(* CoDeSys 2.3 library: ClientStrSock.lib *)
(* Libraries: TcBase.lib 14.5.09 12:14:08, TcSystem.lib 10.9.09 12:54:20, STANDARD.LIB 5.6.98 12:03:02, TcpIp.lib 13.10.11 10:31:34, TcUtilities.lib 17.9.09 15:40:48, TcSocketHelper.lib 20.8.09 10:46:08 *)

(* Global variable list: Global_Variables *)
VAR_GLOBAL CONSTANT
	PLCPRJ_MAX_CONNECTIONS					: UDINT := 5;(* Max. number of server<->client connections *)
	PLCPRJ_SERVER_RESPONSE_TIMEOUT		: TIME 	:= T#500ms;
	PLCPRJ_CLIENT_SEND_CYCLE_TIME			: TIME 	:= T#500ms;

	PLCPRJ_RECEIVER_POLLING_CYCLE_TIME		: TIME 	:= T#200ms;
	PLCPRJ_BUFFER_SIZE						: UDINT := 1000;(* Max. internal fifo/receiver buffer size *)

	(* Some project specific error codes *)
	PLCPRJ_ERROR_RECEIVE_BUFFER_OVERFLOW	: UDINT := 16#8101; (* receive fifo/buffer overflow*)
	PLCPRJ_ERROR_SEND_BUFFER_OVERFLOW		: UDINT := 16#8102;(* send fifo/buffer overflow *)
	PLCPRJ_ERROR_RESPONSE_TIMEOUT			: UDINT := 16#8103;(* receive timeout error *)

	MSG_HEADER 									: STRING(10) :=	'#STR.HEAD#';
	MSG_DATA 										: STRING(10) :=  	'#STR.DATA#';

	MSG_TYPE_SET									: STRING(10) :=	'SET0000000'		;
	MSG_TYPE_RESET								: STRING(10) :=	'RESET00000'	;
	MSG_TYPE_MONITORING							: STRING(10) := 	'MONITOR000'	;

	MSG_SYSTEM_TYPE_1							: STRING(10) := 	'LIGHT00000'	;
	MSG_SYSTEM_TYPE_2							: STRING(10) := 	'ENERGY0000'	;
	MSG_SYSTEM_TYPE_3							: STRING(10) := 	'LEAKAGE000'	;
	MSG_SYSTEM_TYPE_4							: STRING(10) :=	'CLIMATE000'	;

	MSG_DATA_TYPE_1DIGIT							: STRING(10) := 	'1DIG000000'	;
	MSG_DATA_TYPE_3DIGIT							: STRING(10) := 	'3DIG000000'	; (* данные отмасштабированы в пределах 0-255 по шкале 0-100*)
	MSG_DATA_TYPE_4DIGIT							: STRING(10) := 	'4DIG000000'	;
	MSG_DATA_TYPE_8DIGIT							: STRING(10) := 	'8DIG000000'	;
	MSG_DATA_TYPE_S								: STRING(10) :=	'STRING0000'	;

	ARR_DATA_SIZE_1D								: INT := 128;
	ARR_DATA_SIZE_3D								: INT := 32;
	ARR_DATA_SIZE_4D								: INT := 32;
	ARR_DATA_SIZE_8D								: INT := 16;
	ARR_DATA_SIZE_S								: INT := 128;

	TO_SEND										:BYTE:=4;
	TO_RECEIVE									:BYTE :=128;

(*
header
msgMsgType  		= get_buffer_string(strData, 10);
    msgSystemType 		= get_buffer_string(strData, 10);
    msgDeviceType		= get_buffer_string(strData, 10);
    msgDevNum 			= get_buffer_string(strData, 10);
    msgDataType 		= get_buffer_string(strData, 10);
    msgDevision 		= get_buffer_string(strData, 10);
    msgSubDev	 		= get_buffer_string(strData, 10);
    msgReserved_1 		= get_buffer_string(strData, 10);
    msgReserved_2 		= get_buffer_string(strData, 10);
dataheader
*)
(*

MSG_HEADER 				= '#STR.HEAD#'	;
MSG_DATA 				= '#STR.DATA#'	;

MSG_TYPE_SET				= 'SET'		;
MSG_TYPE_RESET				= 'RESET'	;
MSG_TYPE_MONITORING			= 'MONITOR'	;

MSG_SYSTEM_TYPE_1			= 'LIGHT'	;
MSG_SYSTEM_TYPE_2			= 'ENERGY'	;
MSG_SYSTEM_TYPE_3			= 'LEAKAGE'	;
MSG_SYSTEM_TYPE_4			= 'CLIMATE'	;

MSG_DATA_TYPE_1DIGIT			= '1DIG'	;
MSG_DATA_TYPE_3DIGIT			= '3DIG'	;
MSG_DATA_TYPE_4DIGIT			= '4DIG'	;
MSG_DATA_TYPE_150DIGIT			= 'STRING'	;

*)
END_VAR
VAR_GLOBAL
	random		: DRAND := (seed := 10);(* random number generator *)
END_VAR

(* POU F_ADSLOGERROR, ST *)
FUNCTION F_ADSLOGERROR : DINT
(* This function logs communication error messages to the TwinCAT System Log View *)
VAR_INPUT
	sPrefix		: STRING(20);(* Debug message prefix string (allows the identification of log message source) *)
	nErrID		: DWORD; (* Error code *)
END_VAR
IF nErrId = 0 THEN
	F_ADSLOGERROR := ADSLOGSTR( ADSLOG_MSGTYPE_HINT OR ADSLOG_MSGTYPE_LOG, CONCAT( sPrefix, ' No error!   %s'),'' );
ELSIF (  nErrId AND DWORD#16#80000000 ) = 16#80000000 THEN
	F_ADSLOGERROR := ADSLOGDINT( ADSLOG_MSGTYPE_ERROR OR ADSLOG_MSGTYPE_LOG, CONCAT( sPrefix, ' Win32 error: %d' ), SCODE_CODE( nErrId ) );
ELSIF (nErrId AND 16#00008100) =16#00008100 THEN
	F_ADSLOGERROR := ADSLOGDINT( ADSLOG_MSGTYPE_ERROR OR ADSLOG_MSGTYPE_LOG, CONCAT( sPrefix, ' Internal PLC sample project (user) error: %d' ), nErrId );
ELSIF (nErrId AND 16#00008000) =16#00008000 THEN
	F_ADSLOGERROR := ADSLOGDINT( ADSLOG_MSGTYPE_ERROR OR ADSLOG_MSGTYPE_LOG, CONCAT( sPrefix, ' Internal TCP/IP Connection Server error: %d' ), nErrId );
ELSE
	F_ADSLOGERROR := ADSLOGDINT( ADSLOG_MSGTYPE_ERROR OR ADSLOG_MSGTYPE_LOG, CONCAT( sPrefix, ' TwinCAT System error: %d' ), nErrId );
END_IF
END_FUNCTION

(* POU SCODE_CODE, ST *)
FUNCTION SCODE_CODE : DWORD
(* Helper function: returns the lower word of error code *)
VAR_INPUT
	sc		: UDINT;
END_VAR
SCODE_CODE := 16#FFFF AND UDINT_TO_DWORD( sc );
END_FUNCTION

(* POU F_ADSLOGSTRING, ST *)
FUNCTION F_ADSLOGSTRING : DINT
(* This function logs message string to the TwinCAT System Log View *)
VAR_INPUT
	sPrefix	: STRING(20);(* Debug message prefix string (allows the identification of log message source) *)
	sMsg	: T_MaxString;(* Message string *)
END_VAR
VAR
END_VAR
F_ADSLOGSTRING := ADSLOGSTR( ADSLOG_MSGTYPE_HINT OR ADSLOG_MSGTYPE_LOG, CONCAT( sPrefix, '%s' ), sMsg );
END_FUNCTION

(* POU F_DataPrep, ST *)
FUNCTION F_DataPrep : T_MaxString
VAR_INPUT
	msgheader			:STRING(10);
	msgMsgType  		:STRING(10);
	msgSystemType 		:STRING(10);
	msgDeviceType		:STRING(10);
    	msgDevNum 			:STRING(10);
    	msgDataType 		:STRING(10);
    	msgDevision 			:STRING(10);
    	msgSubDev	 		:STRING(10);
    	msgReserved_1 		:STRING(10);
    	msgReserved_2 		:STRING(10);
	dataheader			:STRING(10);
	data1dig				: ARRAY[0..ARR_DATA_SIZE_1D] OF INT;
	data3dig				: ARRAY[0..ARR_DATA_SIZE_3D] OF INT;
	data3dig_Htr			: INT:=255;
	data3dig_Ltr			: INT:=0;
	data4dig				: ARRAY[0..ARR_DATA_SIZE_4D] OF INT;
	data8dig				: ARRAY[0..ARR_DATA_SIZE_8D] OF DINT;
	dataS				: STRING(128);


END_VAR
VAR
	i,j : INT;
	str: T_MaxString	:= '';
	str2: STRING(128) := '';
	str3: STRING(3)	:= '10';
	value:  DINT;
END_VAR
str:= CONCAT(str, msgheader);
str:= CONCAT(str, msgMsgType);
str:= CONCAT(str, msgSystemType);
str:= CONCAT(str, msgDeviceType);
str:= CONCAT(str, msgDevNum);
str:= CONCAT(str, msgDataType);

str:= CONCAT(str, msgDevision);
str:= CONCAT(str, msgSubDev);
str:= CONCAT(str, msgReserved_1);
str:= CONCAT(str, msgReserved_2);
str:= CONCAT(str, dataheader);

IF msgDataType = MSG_DATA_TYPE_1DIGIT THEN

		FOR i:=0 TO ARR_DATA_SIZE_1D-1 DO
			IF data1dig[i] = 1 THEN
				MEMCPY(ADR(str)+110+i, ADR(str3),1);
			ELSE
				MEMCPY(ADR(str)+110+i, ADR(str3)+1,1);
			END_IF
		END_FOR
		MEMSET(ADR(str)+110+ ARR_DATA_SIZE_1D, 33, 255 - (110+ ARR_DATA_SIZE_1D) ); 	(* заполняем восклицательными знаками остаток сообщения*)
END_IF




IF msgDataType = MSG_DATA_TYPE_3DIGIT THEN
		FOR i:=0 TO ARR_DATA_SIZE_3D-1 DO
			value:= F_ValScale( data3dig[i], data3dig_Htr, data3dig_Ltr);
			str2:= F_ValToStr(value, 3);
			MEMCPY(ADR(str)+110+i*3, ADR(str2), 3);
		END_FOR
		MEMSET(ADR(str)+110+ ARR_DATA_SIZE_3D*3, 33, 255 - (110+ ARR_DATA_SIZE_3D*3) ); 	(* заполняем восклицательными знаками остаток сообщения*)
END_IF




IF msgDataType = MSG_DATA_TYPE_4DIGIT THEN

		FOR i:=0 TO ARR_DATA_SIZE_4D-1 DO
			str2:= F_ValToStr(data4dig[i], 4);
			MEMCPY(ADR(str)+110+i*4, ADR(str2), 4);
		END_FOR
		MEMSET(ADR(str)+110+ ARR_DATA_SIZE_4D*4, 33, 255 - (110+ ARR_DATA_SIZE_4D*4) ); 	(* заполняем восклицательными знаками остаток сообщения*)
END_IF

IF msgDataType = MSG_DATA_TYPE_8DIGIT THEN
		FOR i:=0 TO ARR_DATA_SIZE_8D-1 DO
			str2:= F_ValToStr(data8dig[i], 8);
			MEMCPY(ADR(str)+110+i*8, ADR(str2), 8);
		END_FOR
		MEMSET(ADR(str)+110+ ARR_DATA_SIZE_8D*8, 33, 255 - (110+ ARR_DATA_SIZE_8D*8) ); 	(* заполняем восклицательными знаками остаток сообщения*)
END_IF

IF msgDataType = MSG_DATA_TYPE_S  THEN
		MEMCPY(ADR(str)+110, ADR(dataS), 128); 	(* заполняем восклицательными знаками остаток сообщения*)
		MEMSET(ADR(str)+110+128, 33, 255 - (110+ 128) ); 	(* заполняем восклицательными знаками остаток сообщения*)
END_IF

MEMSET(ADR(str)+255, 0, 1); 	(* ставим 0 в самом конце*)
F_DataPrep:=str;
END_FUNCTION

(* POU F_ValScale, ST *)
FUNCTION F_ValScale : DINT
VAR_INPUT
	value : DINT;
	trs_H: INT;
	trs_L: INT;
END_VAR
VAR
	v: INT;
END_VAR

(*
Функция выдает на выходе значение 0 - 100
Аргументами являются входная переменная и верхнее и нижнее значения диапазона
Если входная переменная больше верхнего предела, на выходе 100
Если меньше нижнего предела 0
*)
IF value>trs_H THEN value:= trs_H; END_IF
IF value<trs_L THEN value:= trs_L; END_IF
F_ValScale:= 67;
F_ValScale:= (value - trs_L)*100 / (trs_H - trs_L);
END_FUNCTION

(* POU F_ValToStr, ST *)
FUNCTION F_ValToStr : STRING
VAR_INPUT
	value: DINT; (* значение, которое необходимо перевести в строку*)
	digit: INT; (* количество разрядов, которое должно быть в строчном представлении. Все "пустые" разряды заполняются 0 *)
END_VAR
VAR
	i		: INT := 0;
	val 		: DINT := 0;
	dig		: INT := 0;
	str1		: STRING;
	str2		: STRING;
	str3		: STRING(3):= '000';
END_VAR
IF value <> 0 THEN
val:= value;
	REPEAT
		val := val / 10;
		dig:= dig+1;
	UNTIL
		val = 0
	END_REPEAT
END_IF

str2:= DINT_TO_STRING(value);

FOR i:=0 TO (digit-dig-1) DO
	MEMCPY(ADR(str1)+i, ADR(str3), 1);
END_FOR

MEMCPY(ADR(str1)+digit-dig, ADR(str2), dig);

F_ValToStr:= str1;
END_FUNCTION

(* POU FB_ClientApplication, ST *)
FUNCTION_BLOCK FB_ClientApplication
(* Sample client application. Adapt this code to match your needs. *)

(*
Этот модуль получился аттавизмом. В исходном варианте (который предоставил Бэкхофф) предполагалось, что пользовательская
обработка сообщений будет располагаться прямо здесь. У меня она находится выше - в основной программе. Оттуда вызыва-
ется функция компановки сообщения F_DataPrep и там же определяется когда вызывать отправку. Бэкхофф расчитывал что
я буду писать это здесь... но не сложилось... Пока разбирался, постепенно отключал все лишнее... и в итоге переписал его в
таком виде, в каком он сейчас. Исходный вид (ну или очень близкий к нему ;) ) приведен в комментированом виде ниже.
*)
VAR_INPUT
	bDbg		: BOOL 			:= TRUE;(* TRUE => Enable debug output, FALSE => Disable *)
	sRemoteHost	: STRING(15)	 	:= '127.0.0.1';
	nRemotePort	: UDINT 			:= 9999;
	bEnable		: BOOL 			:= FALSE;
	bRequest	: BOOL:=FALSE;
	msgToServer	: T_MaxString		:= '';
	state: BYTE;
	send_status_reset	:BOOL := FALSE;
END_VAR
VAR_OUTPUT
	eState		: E_SocketConnectionState := eSOCKET_DISCONNECTED;(* TCP/IP connection state *)
	answer		: T_MaxString		:= '';
	bDataReady	: BOOL:= FALSE;
	receive_ok 	: BOOL := FALSE;
	send_ok 		: BOOL:= FALSE;
END_VAR
VAR
	lengthS1		: INT;
	lengthS2		: INT;
	sToServer	: T_MaxString	:= '';
	sFromServer	: T_MaxString	:= '';
	fbClient		: FB_LocalClient;(* Client data exchange control function block *)
	tx 			: FB_FrameStringFifo;(* Tx fifo *)
	rx 			: FB_FrameStringFifo;(* Rx fifo *)
	errors		: FB_ProtErrorFifo;(* Error fifo *)
	sndTimer	: TON;
	rcvTimer		: TON;
(*	state		: BYTE;(* application state *)*)
END_VAR
(*-------------------------- trigger data exchange -----------------------------------------------*)
(*запускаем модуль клиент, передавая сверху в него параметры....*)
fbClient(  bDbg := bDbg, rx := rx, tx := tx, errors := errors, bEnable := bEnable, sRemoteHost := sRemoteHost, nRemotePort := nRemotePort, eState=>eState, received_string=>answer );

(*IF send_status_reset = TRUE THEN send_ok := FALSE; END_IF*)

CASE state OF
	TO_SEND:
		IF fbClient.eState = eSOCKET_CONNECTED THEN
			sToServer := msgToServer;
			tx.A_AddTail( putValue := sToServer );		(* put string to the tx fifo *)
				send_ok:=FALSE;
				IF tx.bOk THEN(* success *)
					send_ok:=TRUE;
				ELSE
					send_ok:=FALSE;
				END_IF

		END_IF

	TO_RECEIVE:
			receive_ok:= FALSE;
			rx.A_RemoveHead();(* fetch string from rx fifo *)
			IF rx.bOk THEN(* success *)
				sFromServer := rx.getValue;
				(* TODO: Check if the response string == request string *)
				receive_ok:= TRUE;
			ELSE
				receive_ok:= FALSE;
			END_IF
END_CASE







(*--------------------------Simple TCP/IP application-----------------------------------------------*)
(* Данный модуль в
state == 0 сбрасывает таймер отправки  и таймаут приема
state == 1 если подключены, взводим таймер отправки сообщения. Если соединения нет уходим в 0:
Пока таймер не сработал крутимся в этом case. Как только таймер сработал
Сбрасываем его
обновляем строку для отправки
вкладываем строку в tx fifo и если это происходит удачно, сбрасываем таймаут приема и переходим в 2:
в противном случае пишем ошибку и остаемся.
state == 2 
Цикл
(
	вырезаем со сдвигом из fifo буфера самое старое сообщение. Если удачно, то  вероятно getvalue(?)
	каким-то образом копируем его в sFromServer и возвращаемся в 0: .Если неудачно, взводим таймаут на прием
	И до тех пор, пока он не случился, крутимся в этом цикле. Если он случился, (!) непонятно (!) у нас все равно
	не наступает условий для выхода из цикла. Условием выхода является упешное извлечение из fifo(rx.bOk). Очень странно... 
	и в таком виде может быть черевато уходами в себя.
)


*)

(*
CASE state OF
	0:(* init state *)
		sndTimer( IN := FALSE, PT := PLCPRJ_CLIENT_SEND_CYCLE_TIME );
		rcvTimer( IN := FALSE, PT := PLCPRJ_SERVER_RESPONSE_TIMEOUT );
		state := 1;

	1:

		(* send string to server *)
		IF fbClient.eState = eSOCKET_CONNECTED THEN
			sndTimer( IN := TRUE );
			IF sndTimer.Q THEN
				sndTimer( IN := FALSE );

				random( );(* create new random number *)
				(*sToServer := CONCAT( 'Random message from client: ', LREAL_TO_STRING(random.Num) );(* simulate user data (string message) *)*)
				lengthS1:= SIZEOF(msgToServer);
				sToServer := msgToServer;
				lengthS2:= SIZEOF(sToServer);


		(*		sToServer := '1234567890123456789012345678901234567890123456789012345678901234567890123456789012345678901234567890AAAAAAAAAA1234567890123456789012345678901234567890123456789012345678901234567890123456789012345678901234567890BBBBBBBBBB123456789012345678901234567890CCCC';
*)
				tx.A_AddTail( putValue := sToServer );(* put string to the tx fifo *)
				IF tx.bOk THEN(* success *)
					rcvTimer( IN := FALSE );
					state := 2;(* wait for response (ECHO from server) ) *)
				ELSE(* TX fifo overflow => log error *)
					errors.A_AddTail( putError := PLCPRJ_ERROR_SEND_BUFFER_OVERFLOW );
				END_IF

			END_IF
		ELSE
			state := 0;
		END_IF

	2:(* wait for response from server *)
		REPEAT
			rx.A_RemoveHead();(* fetch string from rx fifo *)
			IF rx.bOk THEN(* success *)
				sFromServer := rx.getValue;
				(* TODO: Check if the response string == request string *)


				state := 0;(* repeat send-receive cycle *)
			ELSE
				rcvTimer( IN := TRUE );
				IF rcvTimer.Q THEN(* receive timeout => log error *)
					rcvTimer( IN := FALSE );
					errors.A_AddTail( putError := PLCPRJ_ERROR_RESPONSE_TIMEOUT );
					state := 0;
				END_IF
			END_IF
		UNTIL NOT rx.bOk
		END_REPEAT


END_CASE


(*------------------------------- get error messages from error fifo ------------------------------------------*)
(*Отдельный цикл извлекания со сдвигом ошибок из  fifo*)
(*вероятно, bOk - это флаг опустошения буфера... тогда сказанное выше по поводу опасности
 отменяется. Его можно убрать нах. это пока не нужно.
*)
REPEAT
	errors.A_RemoveHead( bDbg := bDbg );
	IF errors.bOk THEN
		;(* TODO: Implement error handler *)
	END_IF
UNTIL NOT errors.bOk
END_REPEAT


*)
END_FUNCTION_BLOCK

(* POU FB_LocalClient, ST *)
FUNCTION_BLOCK FB_LocalClient
(*
----------------------------
НАЗНАЧЕНИЕ
	Устанавливает связь и следит за ее наличием. Передает сообщения. Проверяет входящие.
---------------------------

---------------
Особенности:
	Меня настораживает работа fifo буферов (rx и tx)
	Если передача более или менее работает, то прием сообщений то глючит, то вообще не работает. 
	Пришлось дописать MEMCPY( ADR(received_string), ADR(buffer),  SIZEOF(received_string) ); и только 
	тогда стало появляться приходящее сообщение в received string.

	С отправкой тоже чудеса. Если открыть один сокет и слать пакет скажем раз в секунду, он всегда доходит.
	Если (как в нашем случае) открыть 4 сокета и раз в 300мс слать разные пакеты, то одни не доходят, а других
	приходит (почему-то) лишнее количество... Причем связано это не с какими-то конкретными пакетами. Если 
	поменять их местами в очередности, или даже перезагрузить конечный контроллер, то доходить будут другие.
	Мне не удалось понять где баг. В первую очередь грешу на fifo, т.к. очевидно что здесь что-то не работает...
	Возможно где-то еще есть сюрпизы. 

---------------
*)


VAR_IN_OUT
	tx 			: FB_FrameStringFifo;(* TX fifo *)
	rx 			: FB_FrameStringFifo;(* RX fifo *)
	errors		: FB_ProtErrorFifo;(* Error message fifo *)
END_VAR
VAR_INPUT
	bDbg		: BOOL 			:= TRUE;(* TRUE => Enable debug output, FALSE => Disable debug output *)
	sRemoteHost	: STRING(15) 		:= '192.168.3.229';(* IP address of remote server *)
	nRemotePort	: UDINT			:= 8888;(* Remote server port *)
	bEnable		: BOOL			:= FALSE;(* TRUE => Enable/connect, FALSE => Disable/disconnect *)
	tReconnect	: TIME 			:= T#45s;(* Try to reconnect after this time *)
(*	bRequest: BOOL:= FALSE;*)
END_VAR
VAR_OUTPUT
	eState		: E_SocketConnectionState := eSOCKET_DISCONNECTED;(* TCP/IP connection state *)
	received_string: T_MaxString;
(*	bDataReady: BOOL:=FALSE;*)
END_VAR
VAR
	fbConnect 	: FB_ClientServerConnection := ( tReconnect := T#45s );(* create/release TCP/IP connection *)
	fbSend		: FB_SocketSend;(* send TCP/IP data *)
	fbReceive	: FB_SocketReceive;(* receive TCP/IP data *)
	state 		: BYTE;(* global state *)
	tx_state 		: BYTE;(* tx state *)
	rx_state 		: BYTE;(* rx state *)
	bDisconnect	: BOOL;(* disconnect flag, if set the socket will be closed *)
	pollTimer	: TON;
	cbReceived	: UDINT;(* count of received data bytes *)
	cbRx		: UDINT;(* byte length of received string *)
	rxFrame		: T_MaxString;
	txFrame		: T_MaxString;
	buffer		: ARRAY[0..PLCPRJ_BUFFER_SIZE] OF BYTE;(* Temp. RX buffer *)
	i			: UDINT;
	bAbort		: BOOL;
	sID			: STRING(20) := '';

	bWaitForAnswer: BOOL:=FALSE;
END_VAR
(*
----------------------------
ОПИСАНИЕ (подробное)
---------------------------
state == 0
Сбрасываем fifo приема, передачи и ошибок. Сбрасываем состояния приема и передачи в 0. 
Сбрасываем кол-во принятых данных в 0. Сбрасываем poll таймер. Переходим в state == 1

state == 1
запускаем функциональный блок fbConnect (видимо устанавливаем подключение) крутимся здесь
пока оно не установится. Когда устанавливается, переходим в 2:
state == 2 
Если дизактивирован блок или клиент отключен(поднят флаг), при условии отсутствия входящих и исходящих данных, переходим в 3:
В противном случае  заходим по очереди в ветвления tx_state, rx_state
		tx_state == 0
		Если клиент подключен, извлекаем из tx fifo txFrame. Запускаем блок fbSend со строкой txFrame и, если удачно (bOk), 
		переходим в 1:
		tx_state == 1
		выключаем флаг исполнения  fbSend и проверяем, закончил ли этот блок исполняться (на отправку вписано 5 секунд), если закончил, уходим в 0:
		если при этом были ошибки, делаем дисконнект.

		rx_state == 0
		Если нет дисконнекта, взводим pollTimer, а когда он срабатывает
		Проверяем, (вроде бы) есть ли свободное место в fifo. Если есть, то сбрасываем таймер и выполняем
		блок fbReceive, после чего переходим в 1:
		rx_state == 1
		выключаем флаг исполнения fbReceive и если он закончил работу(на прием так же 5 сек), переходим в  0: а так же
		если не было ошибок и размер принятых данных > 0 (если же принято меньше, то устанавливаем длительность polTimer нормальной)(если были ошибки  пишем их в error fifo и  делаем дисконнект)
		увеличиваем частоту обработки ветвления rx_state, уменьшая до нуля pollTimer
		увеличиваем общий счетчик принятых данных

 		здесь моя вставка копирования из буфера строки

		Далее начинаем цикл (вроде бы парсинга приходящей строки)
		(
			включаем флаг bAbort
			если общее кол-во принятых данных > 0 
			пробегаемся по каждому байту буфера, сравнивая его с 0
			Если находим 0
			запоминаем размер строки + 1 байт знака конца строки
			копируем из буфера в rxFrame данную строку (а если она не лезет, то копируем сколько влезет)
			пихаем rxFrame в rx fifo
			Если успешно (rx.bOk) то сдвигаем значения в буфере на размер забраной строки
				Если в rx fifo есть еще место под rxFrame выключаем флаг bAbort
			Если были ошибки пишем их в eror fifo и делаем дисконнект

			Выходим из цикла если флаг bAbort включен
		)

state == 3
 выключаем блок fbConect и переходим в 0:
---------------------
*)


CASE state OF
	0:(* init state *)
		rx.A_Reset( bDbg := bDbg );(* reset RX fifo (optional) *)
		tx.A_Reset( bDbg := bDbg );(* reset TX fifo (optional) *)
		errors.A_Reset( bDbg := bDbg );(* reset error fifo (optional) *)
		tx_state 		:= 0;
		rx_state 		:= 0;
		pollTimer( IN := FALSE, PT := PLCPRJ_RECEIVER_POLLING_CYCLE_TIME );
		bDisconnect 	:= FALSE;
		cbReceived 	:= 0;
		state 		:= 1;

	1:(* connect *)
		fbConnect( 	sSrvNetID 		:= '',
					nMode			:= CONNECT_MODE_ENABLEDBG,(* enable debug output *)
					sRemoteHost 	:= sRemoteHost,
					nRemotePort 		:= nRemotePort,
					bEnable			:= bEnable,
					tReconnect		:= tReconnect,
					eState			=> eState );
		IF NOT fbConnect.bBusy THEN

			sID 			:= CONCAT( CONCAT('[', DWORD_TO_HEXSTR(fbConnect.hSocket.handle, 4, FALSE) ), ']' );
			tx.sDesc		:= CONCAT( 'CLI.Tx', sID );
			rx.sDesc 		:= CONCAT( 'CLI.Rx', sID );
			errors.sDesc	:= CONCAT( 'CLI.Err', sID );

			IF NOT fbConnect.bError THEN
				IF eState = eSOCKET_CONNECTED THEN(* we are conencted *)
					(*IF bRequest = TRUE THEN*)
					state := 2;
					(*END_IF*)
				END_IF
			ELSE(* connect error => log error *)
				errors.A_AddTail( putError := fbConnect.nErrId );
			END_IF
		END_IF


	2:(* data exchange state *)
		(*bRequest:= FALSE;
		bWaitForAnswer:= TRUE;*)
		bDisconnect := NOT bEnable OR bDisconnect;(* user/internal disconnect requested? *)
		IF bDisconnect AND (tx_state = 0) AND (rx_state = 0) THEN
			state := 3;(* disconnect *)
		ELSE

			(* send tx data *)
			CASE tx_state OF
				0:
					IF NOT bDisconnect THEN
						tx.A_RemoveHead( bDbg := bDbg, getValue => txFrame );(* remove oldest string entry s*)
						IF tx.bOk THEN(* success *)
							fbSend( bExecute := FALSE );
							fbSend(	sSrvNetID 	:= '',
									hSocket		:= fbConnect.hSocket,
									cbLen		:= LEN( txFrame ) + 1,(* send string inclusive string (null) delimiter! *)
									pSrc		:= ADR( txFrame ),(* address of the string variable *)
									bExecute	:= TRUE,
									tTimeout 		:= T#5s );
							tx_state := 1;
						END_IF
					END_IF
				1:(* wait until send not busy *)
					fbSend( bExecute := FALSE );
					IF NOT fbSend.bBusy THEN
						tx_state := 0;
						IF fbSend.bError THEN(* send error => log error and disconnect *)
							errors.A_AddTail( putError := fbSend.nErrId );
							bDisconnect := TRUE;(* set flag *)
						END_IF
					END_IF
			END_CASE



			(* get rx data *)
			CASE rx_state OF
				0:
				(*IF bWaitForAnswer = TRUE THEN*)

					IF NOT bDisconnect THEN
						pollTimer( IN := TRUE );
						IF pollTimer.Q THEN
							IF rx.cbFree >= SIZEOF(rxFrame) THEN(* check free rx fifo space *)
								pollTimer( IN := FALSE );

								fbReceive( bExecute := FALSE );
								fbReceive( 	sSrvNetId	:= '',
											hSocket		:= fbConnect.hSocket,
											cbLen		:= SIZEOF(buffer),(* - cbReceived,*)
											pDest		:= ADR(buffer), (*+ cbReceived,*)
											bExecute	:= TRUE,
											tTimeout		:= T#5s );
								rx_state := 1;
							END_IF
						END_IF
					END_IF
			(*	END_IF*)
				1:(* wait until receive not busy *)
					fbReceive( bExecute := FALSE );
					IF NOT fbReceive.bBusy THEN
						rx_state := 0;
						IF NOT fbReceive.bError THEN
							IF fbReceive.nRecBytes > 0 THEN
								pollTimer( PT := T#0s );(* increase polling speed *)
								cbReceived := cbReceived + fbReceive.nRecBytes;


									MEMSET(ADR(received_string), 0,  SIZEOF(received_string));
									MEMCPY( ADR(received_string), ADR(buffer),  SIZEOF(received_string) );
									(*bWaitForAnswer:= FALSE;
									bDataReady:= TRUE;*)
(*


*)


								(* parse received bytes and extract strings *)
								REPEAT
									bAbort := TRUE;(* set flag *)
									IF cbReceived > 0 THEN

										(* search for string null delimiter *)
										FOR i:= 0 TO cbReceived - 1 BY 1 DO
											IF buffer[i] = 0 THEN (*  end of string position found *)

												cbRx := i + 1;(* calculate the length of string (inclusive the end delimiter) *)
												MEMCPY( ADR(rxFrame), ADR(buffer), MIN(cbRx, SIZEOF(rxFrame) ) );(* copy string bytes to temp string variable *)

												rx.A_AddTail( bDbg := bDbg, putValue := rxFrame );(* add string to the rx fifo *)
												IF rx.bOk THEN
													MEMMOVE( ADR(buffer), ADR(buffer) + cbRx, cbReceived - cbRx );(* move/shift remaining bytes in buffer *)
													cbReceived := cbReceived - cbRx;(* recalculate the remaining data length *)

													IF rx.cbFree >= SIZEOF(rxFrame) THEN (* check free rx buffer space *)
														bAbort := FALSE;(* reset flag, try to parse the next string *)
													END_IF
												ELSE(* fifo overflow => log error and disconnect *)
													errors.A_AddTail( putError := PLCPRJ_ERROR_RECEIVE_BUFFER_OVERFLOW );
													bDisconnect := TRUE;(* set flag *)
													RETURN;
												END_IF

												EXIT;
											END_IF
										END_FOR

									END_IF (* IF cbReceived > 0 THEN *)

								UNTIL bAbort
								END_REPEAT

							ELSE
								pollTimer( PT := PLCPRJ_RECEIVER_POLLING_CYCLE_TIME );
							END_IF(* IF fbReceive.nRecBytes > 0 THEN *)
						ELSE(* receive error => log error and disconnect *)
							errors.A_AddTail( putError := fbReceive.nErrId );
							bDisconnect := TRUE;(* set flag *)
						END_IF
					END_IF

			END_CASE

		END_IF


	3:(* disconnect *)
		fbConnect( bEnable:= FALSE, eState=>eState );
		IF eState = eSOCKET_DISCONNECTED THEN
			state := 0;
		END_IF


END_CASE
END_FUNCTION_BLOCK

(* POU FB_FrameStringFifo, ST *)
FUNCTION_BLOCK FB_FrameStringFifo
(* Tx/Rx (string data) fifo control function block *)
VAR_INPUT
	sDesc		: STRING(20)	:= 'Unknown';(* Debug message description string (allows the identification of log message source) *)
	bDbg		: BOOL		:= FALSE; (* TRUE => Enable debug output, FALSE => Disable *)
	putValue		: T_MaxString := ''; (* String to add (write) to the buffer *)
END_VAR
VAR_OUTPUT
	bOk			: BOOL; 	 	(* TRUE = New entry added or removed succesfully, FALSE = Fifo overflow or fifo empty *)
	getValue		: T_MaxString := ''; (* String removed (read) from buffer *)
	nCount		: UDINT	:= 0;	(* Number of fifo entries *)
	cbFree		: UDINT := 0;	(* Free buffer space *)
END_VAR
VAR
	buffer		: ARRAY[-3..PLCPRJ_BUFFER_SIZE] OF BYTE;(* Internal buffer memory *)
	fbBuffer 		: FB_StringRingBuffer := (bOverwrite := FALSE);(* Basic (lower level) string buffer control function block *)
END_VAR
;
END_FUNCTION_BLOCK
ACTION A_AddTail:
(* adds new fifo entry *)
fbBuffer.A_AddTail( 	pBuffer:= ADR(buffer), cbBuffer:= SIZEOF(buffer),
					putValue:= putValue, bOk=>bOk, nCount=>nCount );
IF bOk THEN
	cbFree := PLCPRJ_BUFFER_SIZE - fbBuffer.cbSize;(* calculate the free buffer space *)
	IF bDbg THEN(* log message *)
		F_ADSLOGSTRING( CONCAT( sDesc, '<=' ), putValue );
	END_IF
END_IF
END_ACTION
ACTION A_RemoveHead:
(* removes oldest fifo entry *)
fbBuffer.A_RemoveHead( pBuffer:= ADR(buffer), cbBuffer:= SIZEOF(buffer),
						bOk=>bOk, getValue=>getValue, nCount=>nCount );
IF bOk THEN
	cbFree := PLCPRJ_BUFFER_SIZE - fbBuffer.cbSize;(* calculate the free buffer space *)
	IF bDbg THEN(* log message *)
		F_ADSLOGSTRING( CONCAT( sDesc, '=>' ), getValue );
	END_IF
END_IF
END_ACTION
ACTION A_Reset:
(* resets fifo = clears all data *)
fbBuffer.A_Reset( pBuffer:= ADR(buffer), cbBuffer:= SIZEOF(buffer),
				bOk=>bOk, getValue=>getValue, nCount=>nCount );
cbFree := PLCPRJ_BUFFER_SIZE;
END_ACTION

(* POU FB_ProtErrorFifo, ST *)
FUNCTION_BLOCK FB_ProtErrorFifo
(* Protocol error fifo control function block *)
VAR_INPUT
	sDesc		: STRING(20)	:= 'Unknown';(* Debug message description string (allows the identification of message source) *)
	bDbg		: BOOL 		:= FALSE; (* TRUE => Enable debug output, FALSE => Disable *)
	putError		: UDINT 		:= 0; (* Error code to add (write) to the fifo *)
END_VAR
VAR_OUTPUT
	bOk			: BOOL; 	 	(* TRUE = New entry added or removed succesfully, FALSE = Fifo overflow or fifo empty *)
	getError		: UDINT		:= 0; (* Error code get/removed (read) from fifo *)
	nCount		: UDINT		:= 0;	(* Number of fifo entries *)
END_VAR
VAR
	buffer	: ARRAY[-3..20] OF BYTE;(* Internal buffer memory *)
	fbBuffer 	: FB_MemRingBuffer;(* Basic (lower level) buffer control function block *)
END_VAR
;
END_FUNCTION_BLOCK
ACTION A_AddTail:
(* adds new fifo entry *)
fbBuffer.A_AddTail( 	pWrite:= ADR( putError ), cbWrite := SIZEOF( putError ),
					pBuffer:= ADR(buffer), cbBuffer:= SIZEOF(buffer),
					bOk=>bOk, nCount=>nCount );
IF bOk THEN
	IF bDbg THEN(* log message *)
		F_ADSLOGERROR( CONCAT( sDesc, '<=' ), putError );
	END_IF
END_IF
END_ACTION
ACTION A_RemoveHead:
(* removes oldest fifo entry *)
fbBuffer.A_RemoveHead( 	pRead := ADR(getError), cbRead := SIZEOF(getError),
						pBuffer:= ADR(buffer), cbBuffer:= SIZEOF(buffer),
						bOk=>bOk, nCount=>nCount );
END_ACTION
ACTION A_Reset:
(* resets fifo = clears all data *)
fbBuffer.A_Reset( pBuffer:= ADR(buffer), cbBuffer:= SIZEOF(buffer),
				bOk=>bOk, nCount=>nCount );
END_ACTION
